# EPICS substitutions: pgpCamlinkApp/camera_config/ImperxC1921.substitutions
# A simple MODEL substitutions file which preserves macro defaults
# but expands any inluded rbvMonitor.template or other templates.
file ImperxC1921.template
{
	{
		P				= "\$(P)",
		R				= "\$(R)",
		PORT			= "\$(PORT)",
		PWIDTH			= "\$(PWIDTH=TRIG:PULSE:WIDTH)",
		PW_SCALE		= "\$(PW_SCALE=1e6)",
		SerialDisable	= "\$(SerialDisable)"
	}
}
